(* IEC 61131-3 sources: SafeDODiag/SODiagDemo, 3 files *)

(* ---- Types.typ ---- *)
(*Structures of IO_TYPE*)

TYPE
	IoInput_TYPE : 	STRUCT
		ContactorSOModuleOK : BOOL; (*Check if SO card for contactor control is in operational mode*)
		Contactor1EnergizeState : BOOL; (*Check if SO card has physically energized output for contactor coil 1*)
		Contactor2EnergizeState : BOOL; (*Check if SO card has physically energized output for contactor coil 2*)
		EDMDiagCode : UINT; (*Read SF_EDM diagnostic code from safety CPU*)
		FdbkSIModuleOK : BOOL; (*Check if SI card for contactor feedback is in operational mode*)
		Contactor1Fdbk : BOOL; (*Check if contactor 1 is open or closed (TRUE--open; FALSE--closed)*)
		Contactor2Fdbk : BOOL; (*Check if contactor 2 is open or closed (TRUE--open; FALSE--closed)*)
		Contactor1EnergizeCurrentOK : BOOL; (*Check if SO card is sending an expected level of current (50 mA - 500 mA) to energize contactor coil 1*)
		Contactor2EnergizeCurrentOK : BOOL; (*Check if SO card is sending an expected level of current (50 mA - 500 mA) to energize contactor coil 2*)
		ContactorOutputInterlockStates : UINT; (*Read output interlock states from SO card*)
	END_STRUCT;
	IoOutput_TYPE : 	STRUCT
		Contactor1EnergizeRequest : BOOL; (*Request SO card output for contactor coil 1*)
		Contactor2EnergizeRequest : BOOL; (*Request SO card output for contactor coil 2*)
		EDMReset : BOOL; (*Request safety CPU to reset SF_EDM error*)
	END_STRUCT;
	IO_TYPE : 	STRUCT  (*Structure with the input and outputs of the plc used by this task*)
		Input : IoInput_TYPE; (*Structure with the inputs of this task*)
		Output : IoOutput_TYPE; (*Structure with the outputs of this task*)
	END_STRUCT;
END_TYPE

(*Structures of IOSP_TYPE - Signal Processing*)

TYPE
	IOSP_TYPE : 	STRUCT  (*Structure with the input and outputs of the plc used by this task*)
		Input : IoInput_TYPE; (*Structure with the inputs of this task*)
		Output : IoOutput_TYPE; (*Structure with the outputs of this task*)
	END_STRUCT;
END_TYPE

(* ---- Main.st ---- *)
PROGRAM _INIT
	// Essential IO
	SafeContactorFub.pSO_Out_Contactor1	:= ADR(IOSP.Output.Contactor1EnergizeRequest);
	SafeContactorFub.pSO_Out_Contactor2	:= ADR(IOSP.Output.Contactor2EnergizeRequest);
	SafeContactorFub.pSO_In_SafeModuleOK			:= ADR(IOSP.Input.ContactorSOModuleOK);
	SafeContactorFub.pSO_In_Output1PhysicalState	:= ADR(IOSP.Input.Contactor1EnergizeState);
	SafeContactorFub.pSO_In_Output2PhysicalState	:= ADR(IOSP.Input.Contactor2EnergizeState);

	(*##################################################
	This fub has four monitoring options, ordered by priority below:
	1) SF_EDM DiagCode from safety CPU (highest priority)
	2) external contactor state monitoring (using SafeDigitalInput0x from SI card)
	3) internal contactor wiring monitoring (using CurrentOK0x from SO card) (lowest priority)
	4) output interlock state monitoring (using FBK_Status_1 from SO card) (independent from and supplementing other monitor options)
	If more than one monitoring options are enabled, the highest priority option will be used by the fub to evaluate contactor open/close behavior.
	##################################################*)

	// These inputs are required by DiagCode monitor and feedback monitor
	SafeContactorFub.pSI_In_SafeModuleOK	:= ADR(IOSP.Input.FdbkSIModuleOK);
	SafeContactorFub.pSI_In_Contactor1Fdbk	:= ADR(IOSP.Input.Contactor1Fdbk);
	SafeContactorFub.pSI_In_Contactor2Fdbk	:= ADR(IOSP.Input.Contactor2Fdbk);

	// These inputs are required by DiagCode monitor
//	SafeContactorFub.Config.CfgDiagCode.EnableMon	:= TRUE;
	SafeContactorFub.Config.DiagCode.StartDelayTime	:= T#2s;	// fub default is 3s but it can be adjusted during fub call like this
	SafeContactorFub.Config.DiagCode.ResetDelayTime	:= T#500ms;	// fub default of 1s may be too longer, so this example uses a shorter delay
	SafeContactorFub.pSF_In_DiagCode				:= ADR(IOSP.Input.EDMDiagCode);

	// These inputs are required by DiagCode monitor and feedback monitor
//	SafeContactorFub.Config.CfgFdbk.EnableMon		:= TRUE;
	SafeContactorFub.Config.Fdbk.StartDelayTime		:= T#2s;	// fub default is 3s but it can be adjusted during fub call like this
	SafeContactorFub.Config.Fdbk.MonitorTime		:= T#200ms;		// no fub default; a value needs to be specified

	// These inputs are required by current OK monitor
//	SafeContactorFub.Config.CfgCurrent.EnableMon	:= TRUE;
	SafeContactorFub.pSO_In_Output1CurrentOK		:= ADR(IOSP.Input.Contactor2EnergizeCurrentOK);
	SafeContactorFub.pSO_In_Output2CurrentOK		:= ADR(IOSP.Input.Contactor2EnergizeCurrentOK);
	SafeContactorFub.Config.Current.MonitorTime		:= T#200ms;	// no fub default; a value needs to be specified

	// These inputs are required by output interlock monitor
//	SafeContactorFub.Config.CfgInterlockState.EnableMon			:= TRUE;
	SafeContactorFub.Config.InterlockState.ChannelPairSelector	:= 1;
	SafeContactorFub.Config.InterlockState.StartDelayTime		:= T#2s;	// fub default is 3s but it can be adjusted during fub call like this
	SafeContactorFub.Config.InterlockState.MonitorTime			:= T#200ms;	// no fub default; a value needs to be specified
	SafeContactorFub.pSO_In_OutputInterlockStates				:= ADR(IOSP.Input.ContactorOutputInterlockStates);

	SafeContactorFub.Cmd.Simulation.EnableSim := DiagCpuIsARsim();
END_PROGRAM

PROGRAM _CYCLIC
	// Read inputs
	brsmemcpy( ADR( IOSP.Input ), ADR( IO.Input ), SIZEOF( IOSP.Input ) );

	IF( bToggleDemoMode )THEN
		// Check for user output request
		SafeDigitalOutFub.Cmd.OutputRequest	:= bRequestOutput;
		// Check for user reset request of SF_EDM error
		SafeDigitalOutFub.Cmd.Reset			:= bReset;
		// Run fub
		SafeDigitalOutFub();
		// Pass through SF_EDM reset request
		IOSP.Output.EDMReset				:= SafeDigitalOutFub.Status.SafetyResetRequested;
	ELSE
		// Check for user output request
		SafeContactorFub.Cmd.OutputRequest	:= bRequestOutput;
		// Check for user reset request of SF_EDM error
		SafeContactorFub.Cmd.Reset			:= bReset;
		// Run fub
		SafeContactorFub();
		// Pass through SF_EDM reset request
		IOSP.Output.EDMReset				:= SafeContactorFub.Status.SafetyResetRequested;
	END_IF

	// Write outputs
	brsmemcpy( ADR( IO.Output ), ADR( IOSP.Output ), SIZEOF( IOSP.Output ) );
END_PROGRAM

PROGRAM _EXIT
END_PROGRAM

(* ---- Variables.var ---- *)
VAR
	bRequestOutput : BOOL;
	bReset : BOOL;
	bToggleDemoMode : BOOL;
	SafeContactorFub : SContactor;
	SafeDigitalOutFub : SDigitalOut;
	IO : IO_TYPE;
	IOSP : IOSP_TYPE;
END_VAR
